Staubli VAL3: loadPoint.pgx

public program loadPoint(string x_sItem, num& x_nResult)
  local string l_sType
  local string l_sMessage
  local num l_nResult
begin
  //
  // !!! REMOVE DUE PROBLEMS of CROSS LINK
  //
  //  // load the select trajectory..already loaded
  //  call getTrajType(l_sType)
  //  if find(pPoint:libPath(),saveData:sPathTraj)==-1
  //    l_nResult=pPoint:libLoad(saveData:sPathTraj+"POINT")
  //    delay(0)
  //    if saveData:bDebug
  //      ? "HOME loading POINT..."+saveData:sPathTraj+"POINT"+toString("",l_nResult)
  //    endIf
  //  endIf
  //  if isDefined(pPoint:tTraj[x_sItem])
  //    // validate
  //    x_nResult=0
  //  elseIf x_sItem!=""
  //    // not FOUND
  //    call language:message(l_sMessage,-7)
  //    x_nResult=-1
  //    popUpMsg(l_sMessage+x_sItem)
  //  endIf
end
